8: (*промывка чистой водой после дезинфекции, ожидание протока на возврате*)
  PastPrev:=Step;
  q_SP_P1:=i_PumpCapacity;
  StepBackPump:=1; (*включен возврат и контроль возврата*)

  Start_Control_Q4 := TRUE; (*контроль потока в танк возвратной воды Q4 *)
  ModeControl_Q5 := 2; (*поддержание уровня в цирк баке при промывке и вытесн через цирк бак, контроль насоса Р1*)

  IF Return_OK THEN (*возврта в норме*)
      T_Process.PT:=DINT_TO_TIME(i_TimeSwill*60000);
     Step:=9;
  END_IF;

  q_VisuMode:=19;

9: (*промывка чистой водой после дезинфекции - отсчет времени*)
  PastPrev:=Step;
  q_SP_P1:=i_PumpCapacity;
  StepBackPump:=1; (*включен возврат и контроль возврата*)

  Start_Control_Q4 := TRUE; (*контроль потока в танк возвратной воды Q4 *)
  ModeControl_Q5 := 2; (*поддержание уровня в цирк баке при промывке и вытесн через цирк бак, контроль насоса Р1*)


     (*расчет времени для визуализ*)
    q_Vis_tim_Process := TRUE; (*визуализация полей времени*)
    Last_Time_min := (TIME_TO_DINT(T_Process.PT-T_Process.ET))/60000 ;
    Last_Time_sec := (TIME_TO_DINT(T_Process.PT-T_Process.ET)/1000) - Last_Time_min * 60 ;

   T_Process.in:=TRUE;
   IF T_Process.Q THEN
      T_Process.in:=FALSE;
      Step:=10;
   END_IF;

  q_VisuMode:=19;

10: (*опустошение цирк бака*)
  PastPrev:=Step;
  q_VA51:=TRUE;
  q_P1:=TRUE;
  q_SP_P1:=i_PumpCapacity;
  StepBackPump:=1; (*включен возврат и контроль возврата*)

  Start_Control_Q4 := TRUE; (*контроль потока в танк возвратной воды Q4 *)


    IF (T_LSL_off.Q AND NOT i_LSM) THEN  (*циркуляционный бак пустой*)
      StepBackPump:=3;
      T_Delay.IN:= FALSE;
      Step:=11 ;
    END_IF;

  q_VisuMode:=4;

11: (*откачка из маршрута*)
  PastPrev:=Step;
  StepBackPump:=3; (*откачка из маршрута*)

  T_Delay.PT:=DINT_TO_TIME(i_TimeDelay*1000); (*задержка закрытия клапана*)
  T_Delay.IN:=TRUE;
  q_VA51:=NOT T_Delay.Q ;

  Start_Control_Q4 := TRUE; (*контроль потока в танк возвратной воды Q4 *)


      IF EndReturn  THEN (*докачали из маршрута*)
          T_Delay.IN:= FALSE;
         StepBackPump:=0; (*выключить возврат и контроль возврата*)
         Step:=12;
      END_IF;

  q_VisuMode:=4;

12: (*выполнено*)
  q_VisuMode:=1;
  StepBackPump := 0; (*выключить вовзрат и контроль возврата*)




(*-----------------авария----------------*)
30: (*авария*)
       q_VisuMode:=11;
       q_Red:=TRUE;
       q_Sirena :=TRUE;
       T_Process.IN := FALSE; (*остановка таймера процесса*)
       IF AlarmReset AND (PastPrev=4 OR PastPrev=9)  THEN
          T_Process.PT := DINT_TO_TIME(Last_Time_min*60000 + Last_Time_sec*1000);  (*уставка для таймера  в случае выхода в аварию*)
          Step := PastPrev;
       ELSIF AlarmReset AND PastPrev<>4 AND PastPrev<>9 THEN
          Step := PastPrev;
       END_IF;

(*-----------------пауза----------------*)
35: (*пауза*)
       q_VisuMode:=12;
       q_Yellow:=TRUE;
       T_Process.IN := FALSE; (*остановка таймера процесса*)
       IF NOT i_Pause AND (PastPrev=4 OR PastPrev=9)  THEN
          T_Process.PT := DINT_TO_TIME(Last_Time_min*60000 + Last_Time_sec*1000);  (*уставка для таймера  в случае выхода в аварию*)
          Step := PastPrev;
       ELSIF NOT i_Pause AND PastPrev<>4 AND PastPrev<>9 THEN
          Step := PastPrev;
       END_IF;

(*-----------------пауза - не готов маршрут----------------*)
36: (*пауза*)
       q_VisuMode:=18;
       q_Yellow:=TRUE;
       T_Process.IN := FALSE; (*остановка таймера процесса*)
       IF i_Ready_Route AND (PastPrev=4 OR PastPrev=9)  THEN
          T_Process.PT := DINT_TO_TIME(Last_Time_min*60000 + Last_Time_sec*1000);  (*уставка для таймера  в случае выхода в аварию*)
          Step := PastPrev;
       ELSIF i_Ready_Route AND PastPrev<>4 AND PastPrev<>9 THEN
          Step := PastPrev;
       END_IF;


 END_CASE;

(*блок поддержания уровня в циркуляционном баке во время мойки и при откачке*)
Control_Q5(
	i_P1:= q_P1,
	i_VA551:= q_VA551 ,
	i_VA11:= q_VA11 ,
	i_VA51:= q_VA51 ,
	i_LSL:= i_LSL ,
	i_LSM:= i_LSM ,
	i_LSH:= i_LSH ,
	i_RouteType:= i_RouteType,
	i_Time_LSH_on:= i_Time_LSH_on ,
	i_Time_LSM_on:= i_Time_LSM_on ,
	i_Time_LSM_off:= i_Time_LSM_off ,
	i_Time_LSL_off:= i_Time_LSL_off ,
	i_TimeDelay:= i_TimeDelay ,
	i_ModeControl_Q5:= ModeControl_Q5 ,
	i_StepBackPump:= StepBackPump ,
	q_P1=> q_P1 ,
	q_VA551=> q_VA551 ,
	q_VA11=> q_VA11 ,
	q_VA51=> q_VA51 ,
	q_Alarm_Empty_Q5=> q_Alarm_Empty_Q5 ,
	q_StepBackPump=> StepBackPump);

(*блок контроля и управления возвратом моющих средств*)
Return_Flow(
	i_AlarmPause:= (Step>=30),  (*в аварии или в паузе мойки или неготовности маршрута*)
	i_FS:= i_FS ,
	i_StepBackPump:= StepBackPump ,
	i_RouteType:= i_RouteType ,
	i_Current_VolumeFC11:= i_Current_VolumeFC11 ,
	i_TimeDelayRetPump:= i_TimeDelayRetPump ,
	i_TimeDelayRetFlow:= i_TimeDelayRetFlow ,
	i_TimeAlarmBackFlow:= i_TimeAlarmBackFlow ,
	q_BackPump=> q_BackPump ,
	q_AlarmBackFlow=> q_AlarmBackFlow ,
	q_EndReturn=>EndReturn  ,
      q_Return_OK=>Return_OK ,
	q_ZeroCount_FC11=> q_ZeroCount_FC11 ,
	q_FC11_start=> q_FC11_start );

(*блок контроля потока в танк возвратной воды Q4*)
Control_Q4(
	i_Start:= Start_Control_Q4 ,
	i_Block_Q4_in:= i_Block_Q4_in ,
	i_VA401:= q_VA401 ,
	i_VA541:= q_VA541 ,
	i_TimeDelay:= i_TimeDelay ,
	q_VA401=> q_VA401 ,
	q_VA541=> q_VA541);


T_Process();
T_Delay();
T_LSH_on (IN:=i_LSH,     PT:=DINT_TO_TIME(i_Time_LSH_on*1000));
T_LSM_on (IN:=i_LSM,     PT:=DINT_TO_TIME(i_Time_LSM_on*1000));
T_LSM_off(IN:=NOT i_LSM, PT:=DINT_TO_TIME(i_Time_LSM_off*1000));
T_LSL_off(IN:=NOT i_LSL, PT:=DINT_TO_TIME(i_Time_LSL_off*1000));
END_FUNCTION_BLOCK

(* POU Inputs, ST *)
PROGRAM Inputs  (*блок масштабирования и обработки аналоговых величин*)
VAR
(*-----общие----*)
	fb_TE2  :AnScaling;
	fb_TE3  :AnScaling;
	fb_LE1  :AnScaling;
	fb_LE2  :AnScaling;
	fb_LE3  :AnScaling;
	fb_LE4  :AnScaling;
	fb_TE4  :AnScaling;

(*---контур 1---*)
	fb_TE11:AnScaling;
	fb_PE1  :AnScaling;
	fb_FE1  :AnScaling;
	fb_QE1  :AnScaling;
	fb_TE21 :AnScaling;

(*---контур 2---*)
	fb_TE12 :AnScaling;
	fb_PE2  :AnScaling;
	fb_FE2  :AnScaling;
	fb_QE2  :AnScaling;
	fb_TE22 :AnScaling;


(*расчет концентрации растворов*)
    Conc_C1 :Concentrat_Mode;
    Conc_C2 :Concentrat_Mode;


END_VAR
(*-----------Общие датчики-------------*)
fb_TE2(
	i_IW_an:=		TE2_i ,
	i_SensorType:=	1 ,
	i_An_Scale:=	An_Scale_TE2 ,
	q_Error=>		Error_TE2 ,
	q_LE=>			i_TE2 );

fb_TE3(
	i_IW_an:=		TE3_i ,
	i_SensorType:=	1 ,
	i_An_Scale:=	An_Scale_TE3 ,
	q_Error=>		Error_TE3 ,
	q_LE=>			i_TE3 );

fb_LE1(
	i_IW_an:=		LE1_i ,
	i_SensorType:=	0 ,
	i_An_Scale:=	An_Scale_LE1 ,
	q_Error=>		Error_LE1 ,
	q_LE=>			i_LE1 );

fb_LE2(
	i_IW_an:=		LE2_i ,
	i_SensorType:=	0 ,
	i_An_Scale:=	An_Scale_LE2 ,
	q_Error=>		Error_LE2 ,
	q_LE=>			i_LE2 );

fb_LE3(
	i_IW_an:=		LE3_i ,
	i_SensorType:=	0 ,
	i_An_Scale:=	An_Scale_LE3 ,
	q_Error=>		Error_LE3 ,
	q_LE=>			i_LE3 );



(*раскомментировать при использовании танка возвратной воды Q4*)
(*
fb_LE4(
	i_IW_an:=		LE4_i ,
	i_SensorType:=	0 ,
	i_An_Scale:=	An_Scale_LE4 ,
	q_Error=>		Error_LE4 ,
	q_LE=>			i_LE4 );

fb_TE4(
	i_IW_an:=		TE4_i ,
	i_SensorType:=	1 ,
	i_An_Scale:=	An_Scale_TE4 ,
	q_Error=>		Error_TE4 ,
	q_LE=>			i_TE4 );

*)

(*------------------------------Контур 1---------------------------*)

fb_TE11(
	i_IW_an:=		TE11_i ,
	i_SensorType:=	1 ,
	i_An_Scale:=	An_Scale_TE11 ,
	q_Error=>		Error_TE11 ,
	q_LE=>			i_TE11);

fb_PE1(
	i_IW_an:=		PE1_i ,
	i_SensorType:=	1 ,
	i_An_Scale:=	An_Scale_PE1 ,
	q_Error=>		Error_PE1 ,
	q_LE=>			i_PE1 );
IF i_PE1<0 THEN
   i_PE1:=0;
END_IF;

fb_FE1(
	i_IW_an:=		FE1_i ,
	i_SensorType:=	1 ,
	i_An_Scale:=	An_Scale_FE1 ,
	q_Error=>		Error_FE1 ,
	q_LE=>			i_FE1 );


fb_QE1(
	i_IW_an:=		QE1_i ,
	i_SensorType:=	1 ,
	i_An_Scale:=	An_Scale_QE1 ,
	q_Error=>		Error_QE1 ,
	q_LE=>			i_QE1 );


fb_TE21(
	i_IW_an:=		TE21_i ,
	i_SensorType:=	1 ,
	i_An_Scale:=	An_Scale_TE21 ,
	q_Error=>		Error_TE21 ,
	q_LE=>			i_TE21);



(*------------------------------Контур 2---------------------------*)
fb_TE12(
	i_IW_an:=		TE12_i ,
	i_SensorType:=	1 ,
	i_An_Scale:=	An_Scale_TE12 ,
	q_Error=>		Error_TE12 ,
	q_LE=>			i_TE12);


fb_PE2(
	i_IW_an:=		PE2_i ,
	i_SensorType:=	1 ,
	i_An_Scale:=	An_Scale_PE2 ,
	q_Error=>		Error_PE2 ,
	q_LE=>			i_PE2 );
IF i_PE2<0 THEN
   i_PE2:=0;
END_IF;

fb_FE2(
	i_IW_an:=		FE2_i ,
	i_SensorType:=	1 ,
	i_An_Scale:=	An_Scale_FE2 ,
	q_Error=>		Error_FE2 ,
	q_LE=>			i_FE2 );

fb_QE2(
	i_IW_an:=		QE2_i ,
	i_SensorType:=	1 ,
	i_An_Scale:=	An_Scale_QE2 ,
	q_Error=>		Error_QE2 ,
	q_LE=>			i_QE2 );

fb_TE22(
	i_IW_an:=		TE22_i ,
	i_SensorType:=	1 ,
	i_An_Scale:=	An_Scale_TE22 ,
	q_Error=>		Error_TE22 ,
	q_LE=>			i_TE22);


(*--------------Расчет концентрации растворов------------*)
Conc_C1(
	i_QE:=i_QE1 ,
	i_TE:=i_TE21 ,
	i_ModeQE:=ModeQE_C1 ,
	q_QE_priv=>QE1_priv ,
	q_QE=>QE1 );

Conc_C2(
	i_QE:=i_QE2 ,
	i_TE:=i_TE22 ,
	i_ModeQE:=ModeQE_C2 ,
	q_QE_priv=>QE2_priv ,
	q_QE=>QE2 );
END_PROGRAM

(* POU Concentrat_Mode, ST *)
FUNCTION_BLOCK Concentrat_Mode
VAR_INPUT
	i_QE		: REAL;
	i_TE		: REAL;
	i_ModeQE	: INT;
END_VAR
VAR_OUTPUT
	q_QE_priv	: REAL;
	q_QE		: REAL;

END_VAR
VAR
END_VAR
CASE i_ModeQE OF    (*выбор пересчета по контуру*)

0:(*-------------Расчет концентрации щелочи-----------------*)
q_QE_priv:=i_QE/(1+Koef_tempAlk*(i_TE-Temp_etalonAlk));  (*приведение проводимости к эталонной*)
q_QE := 0.5+(q_QE_priv-QE_null_Alk)/Psi_Alk;   (*расчет концентрации %*)

1:(*-------------Расчет концентрации кислоты-----------------*)
q_QE_priv:=i_QE/(1+Koef_tempAcid*(i_TE-Temp_etalonAcid));  (*приведение проводимости к эталонной*)
q_QE := 0.5+(q_QE_priv-QE_null_Acid)/Psi_Acid;   (*расчет концентрации %*)

END_CASE;

IF q_QE_priv<0 THEN
   q_QE_priv:=0;
END_IF;


IF q_QE<0 THEN
   q_QE:=0;
END_IF;
END_FUNCTION_BLOCK

(* POU AlarmReaction, ST *)
PROGRAM AlarmReaction
VAR
	T_PS   :TON;      (*таймер аварии сжатого воздуха*)
	T_FE11 :TON;      (*таймер аварии протока на подаче*)
	T_FE12 :TON;      (*таймер аварии протока на подаче*)

END_VAR
(*авария низкого давления сжатого воздуха с таймером*)
   T_PS.IN := NOT PS1_i;
IF T_PS.Q THEN
  	Alarm_PS := TRUE;
END_IF;
IF PS1_i AND Alarm_PS AND AlarmReset THEN
   Alarm_PS := FALSE;
END_IF;
T_PS(PT:=T#3s);

(*авария макс давления PE1*)
IF i_PE1>MaxPressure_C1 THEN
   Alarm_PE1 := TRUE;
ELSIF i_PE1<(MaxPressure_C1-2.0) AND  Alarm_PE1 AND AlarmReset THEN
   Alarm_PE1 := FALSE;
END_IF;

(*авария макс давления PE2*)
IF i_PE2>MaxPressure_C2 THEN
   Alarm_PE2 := TRUE;
ELSIF i_PE2<(MaxPressure_C2-2.0) AND  Alarm_PE2 AND AlarmReset THEN
   Alarm_PE2 := FALSE;
END_IF;


(*аварийный стоп*)
IF NOT AlarmStop_i THEN
   Alarm_Stop:=TRUE;
ELSIF Alarm_Stop AND AlarmReset THEN
   Alarm_Stop:=FALSE;
END_IF;

(*нет протока на подаче контура 1*)
T_FE11.IN:=w_qDevice_C1.P1 AND SP_P1>1500 AND i_FE1<1500;
IF T_FE11.Q THEN
   Alarm_FE11:=TRUE;
END_IF;
T_FE11(PT:= DINT_TO_TIME(Time_Alarm_FE*1000));

(*нет протока на подаче контура 2*)
T_FE12.IN:=w_qDevice_C2.P1 AND SP_P2>1500 AND i_FE2<1500;
IF T_FE12.Q THEN
   Alarm_FE12:=TRUE;
END_IF;
T_FE12(PT:= DINT_TO_TIME(Time_Alarm_FE*1000));



IF AlarmReset THEN
   Alarm_FE11:=FALSE;
   Alarm_FE12:=FALSE;
   AlarmBackFlow_C1:=FALSE;
   AlarmBackFlow_C2:=FALSE;
   HeatingAlarm_C1:=FALSE;
   HeatingAlarm_C2:=FALSE;
   CondAlarm_C1:=FALSE;
   CondAlarm_C2:=FALSE;
   Alarm_Empty_Q5:=FALSE;
   Alarm_Empty_Q6:=FALSE;
END_IF;


(*аварийный уровень в баке концентрата кислоты*)
IF NOT LS81_i THEN
   Alarm_LS81:= TRUE;
ELSE
   Alarm_LS81:= FALSE;
END_IF;
(*низкий уровень в баке концентрата кислоты*)
IF NOT LS82_i THEN
   Alarm_LS82:= TRUE;
ELSE
   Alarm_LS82:= FALSE;
END_IF;

(*аварийный уровень в баке концентрата щелочи*)
IF NOT LS71_i THEN
   Alarm_LS71:= TRUE;
ELSE
   Alarm_LS71:= FALSE;
END_IF;
(*низкий уровень в баке концентрата щелочи*)
IF NOT LS72_i THEN
   Alarm_LS72:= TRUE;
ELSE
   Alarm_LS72:= FALSE;
END_IF;



(*минимальный уровень в танке чистой воды*)
IF i_LE1<MinAlarmLevel_Q1 THEN
   Alarm_MinLev_Q1:=TRUE;
ELSIF Alarm_MinLev_Q1 AND i_LE1>(MinAlarmLevel_Q1+5.0) AND AlarmReset THEN
   Alarm_MinLev_Q1:=FALSE;
END_IF;

(*минимальный уровень в танке щелочи*)
IF i_LE2<MinAlarmLevel_Q2 THEN
   Alarm_MinLev_Q2:=TRUE;
ELSIF Alarm_MinLev_Q2 AND i_LE2>(MinAlarmLevel_Q2+5.0) AND AlarmReset THEN
   Alarm_MinLev_Q2:=FALSE;
END_IF;

(*минимальный уровень в танке кислоты*)
IF i_LE3<MinAlarmLevel_Q3 THEN
   Alarm_MinLev_Q3:=TRUE;
ELSIF Alarm_MinLev_Q3 AND i_LE3>(MinAlarmLevel_Q3+5.0) AND AlarmReset THEN
   Alarm_MinLev_Q3:=FALSE;
END_IF;
END_PROGRAM

(* POU DeviceControl, ST *)
PROGRAM DeviceControl
VAR
	Step_Q1		: INT;

(*---блоки управления механизмами--*)
	fb_VA1   	:Valve;
(*контур 1*)
	fb_VA541 	:Valve;
	fb_VA401 	:Valve;
	fb_VA201 	:Valve;
	fb_VA301 	:Valve;
	fb_VA41  	:Valve;
	fb_VA11  	:Valve;
	fb_VA21  	:Valve;
	fb_VA31  	:Valve;
	fb_VA5 		:Valve;
	fb_VA501 	:Valve;
	fb_VA51  	:Valve;
	fb_VA511 	:Valve;
	fb_VA521 	:Valve;
	fb_VA531 	:Valve;
	fb_P1    		:Pump;
(*контур 2*)
	fb_VA642 	:Valve;
	fb_VA402 	:Valve;
	fb_VA202 	:Valve;
	fb_VA302 	:Valve;
	fb_VA42  	:Valve;
	fb_VA12  	:Valve;
	fb_VA22  	:Valve;
	fb_VA32  	:Valve;
	fb_VA6 		:Valve;
	fb_VA602 	:Valve;
	fb_VA62  	:Valve;
	fb_VA612 	:Valve;
	fb_VA622 	:Valve;
	fb_VA632 	:Valve;
	fb_P2    		:Pump;

(*-----ПИД-регуляторы-----*)
	PID_VR1  :PID_M;
	PID_VR2  :PID_M;

	PID_P1   :PID_M;
	PID_P2   :PID_M;

END_VAR
(*управление поддержанием уровня чистой воды в Q1*)
CASE Mode_Q1 OF
0:(*автомат*)
 	CASE Step_Q1 OF
  	0:
   		IF i_LE1<=MinLevel_Q1 THEN
      			Step_Q1:=1;
   		END_IF;
  	1:
   		q_VA1:=TRUE;
   		IF i_LE1>=MaxLevel_Q1 THEN
      			Step_Q1:=0;
   		END_IF;
	END_CASE;
  	Man_VA1:=FALSE;
1:(*ручной*)
  	q_VA1:=Man_VA1;
END_CASE;

fb_VA1(
    i_AlarmReset:=AlarmReset ,
	i_VAopen:=NOT VA1_i ,
	i_VAclose:=VA1_i ,
	i_DiagVA:=DiagVA1 ,
	i_SetVA:=q_VA1 ,
	i_TimerPT:=T#8s ,
	q_Alarm=>Alarm_VA1 ,
	q_VA=>VA1_q);
Mode_VA1:=fb_VA1.Mode;


(*----------------------Управление механизмами с контролем состояния-----------------*)

(*---------------------Контур 1------------------------*)
fb_VA541(
    i_AlarmReset:=AlarmReset ,
	i_VAopen:=NOT VA541_i ,
	i_VAclose:=VA541_i ,
	i_DiagVA:=wDiagVA_C1.VA541 ,
	i_SetVA:=w_qDevice_C1.VA541 ,
	i_TimerPT:=T#5s ,
	q_Alarm=>Alarm_VA541 ,
	q_VA=>VA541_q);
Mode_VA541:=fb_VA541.Mode;

(* раскомментировать при использовании танка возвратной воды Q4
fb_VA401(
    i_AlarmReset:=AlarmReset ,
	i_VAopen:=NOT VA401_i ,
	i_VAclose:=VA401_i ,
	i_DiagVA:=wDiagVA_C1.VA401 ,
	i_SetVA:=w_qDevice_C1.VA401 ,
	i_TimerPT:=T#5s ,
	q_Alarm=>Alarm_VA401 ,
	q_VA=>VA401_q);
Mode_VA401:=fb_VA401.Mode;
*)

fb_VA201(
    i_AlarmReset:=AlarmReset ,
	i_VAopen:=NOT VA201_i ,
	i_VAclose:=VA201_i ,
	i_DiagVA:=wDiagVA_C1.VA201 ,
	i_SetVA:=w_qDevice_C1.VA201 ,
	i_TimerPT:=T#5s ,
	q_Alarm=>Alarm_VA201 ,
	q_VA=>VA201_q);
Mode_VA201:=fb_VA201.Mode;

fb_VA301(
    i_AlarmReset:=AlarmReset ,
	i_VAopen:=NOT VA301_i ,
	i_VAclose:=VA301_i ,
	i_DiagVA:=wDiagVA_C1.VA301 ,
	i_SetVA:=w_qDevice_C1.VA301 ,
	i_TimerPT:=T#5s ,
	q_Alarm=>Alarm_VA301 ,
	q_VA=>VA301_q);
Mode_VA301:=fb_VA301.Mode;

(*раскомментировать при использовании танка возвратной воды Q4
fb_VA41(
    i_AlarmReset:=AlarmReset ,
	i_VAopen:=NOT VA41_i ,
	i_VAclose:=VA41_i ,
	i_DiagVA:=wDiagVA_C1.VA41 ,
	i_SetVA:=w_qDevice_C1.VA41 ,
	i_TimerPT:=T#7s ,
	q_Alarm=>Alarm_VA41 ,
	q_VA=>VA41_q);
Mode_VA41:=fb_VA41.Mode;
*)

fb_VA11(
    i_AlarmReset:=AlarmReset ,
	i_VAopen:=NOT VA11_i ,
	i_VAclose:=VA11_i ,
	i_DiagVA:=wDiagVA_C1.VA11 ,
	i_SetVA:=w_qDevice_C1.VA11 ,
	i_TimerPT:=T#7s ,
	q_Alarm=>Alarm_VA11 ,
	q_VA=>VA11_q);
Mode_VA11:=fb_VA11.Mode;

fb_VA21(
    i_AlarmReset:=AlarmReset ,
	i_VAopen:=NOT VA21_i ,
	i_VAclose:=VA21_i ,
	i_DiagVA:=wDiagVA_C1.VA21 ,
	i_SetVA:=w_qDevice_C1.VA21 ,
	i_TimerPT:=T#7s ,
	q_Alarm=>Alarm_VA21 ,
	q_VA=>VA21_q);
Mode_VA21:=fb_VA21.Mode;

fb_VA31(
    i_AlarmReset:=AlarmReset ,
	i_VAopen:=NOT VA31_i ,
	i_VAclose:=VA31_i ,
	i_DiagVA:=wDiagVA_C1.VA31 ,
	i_SetVA:=w_qDevice_C1.VA31 ,
	i_TimerPT:=T#7s ,
	q_Alarm=>Alarm_VA31 ,
	q_VA=>VA31_q);
Mode_VA31:=fb_VA31.Mode;


fb_VA5(
    i_AlarmReset:=AlarmReset ,
	i_VAopen:=NOT VA5_i ,
	i_VAclose:=VA5_i ,
	i_DiagVA:=wDiagVA_C1.VA5 ,
	i_SetVA:=w_qDevice_C1.VA5 ,
	i_TimerPT:=T#8s ,
	q_Alarm=>Alarm_VA5 ,
	q_VA=>VA5_q);
Mode_VA5:=fb_VA5.Mode;

fb_VA501(
    i_AlarmReset:=AlarmReset ,
	i_VAopen:=NOT VA501_i ,
	i_VAclose:=VA501_i ,
	i_DiagVA:=wDiagVA_C1.VA501 ,
	i_SetVA:=w_qDevice_C1.VA501 ,
	i_TimerPT:=T#5s ,
	q_Alarm=>Alarm_VA501 ,
	q_VA=>VA501_q);
Mode_VA501:=fb_VA501.Mode;

fb_VA51(
    i_AlarmReset:=AlarmReset ,
	i_VAopen:=NOT VA51_i ,
	i_VAclose:=VA51_i ,
	i_DiagVA:=wDiagVA_C1.VA51 ,
	i_SetVA:=w_qDevice_C1.VA51 ,
	i_TimerPT:=T#5s ,
	q_Alarm=>Alarm_VA51 ,
	q_VA=>VA51_q);
Mode_VA51:=fb_VA51.Mode;

fb_VA511(
    i_AlarmReset:=AlarmReset ,
	i_VAopen:=NOT VA511_i ,
	i_VAclose:=VA511_i ,
	i_DiagVA:=wDiagVA_C1.VA511 ,
	i_SetVA:=w_qDevice_C1.VA511 ,
	i_TimerPT:=T#5s ,
	q_Alarm=>Alarm_VA511 ,
	q_VA=>VA511_q);
Mode_VA511:=fb_VA511.Mode;

fb_VA521(
    i_AlarmReset:=AlarmReset ,
	i_VAopen:=NOT VA521_i ,
	i_VAclose:=VA521_i ,
	i_DiagVA:=wDiagVA_C1.VA521 ,
	i_SetVA:=w_qDevice_C1.VA521 ,
	i_TimerPT:=T#5s ,
	q_Alarm=>Alarm_VA521 ,
	q_VA=>VA521_q);
Mode_VA521:=fb_VA521.Mode;

fb_VA531(
    i_AlarmReset:=AlarmReset ,
	i_VAopen:=NOT VA531_i ,
	i_VAclose:=VA531_i ,
	i_DiagVA:=wDiagVA_C1.VA531 ,
	i_SetVA:=w_qDevice_C1.VA531 ,
	i_TimerPT:=T#5s ,
	q_Alarm=>Alarm_VA531 ,
	q_VA=>VA531_q);
Mode_VA531:=fb_VA531.Mode;

(*насос подачи *)
fb_P1(
	i_AlarmReset:= AlarmReset ,
	IsV_P:=w_qDevice_C1.P1 ,
	Protect:= NOT ProtectP1_i ,
	SetV_P:=w_qDevice_C1.P1 ,
	Timer_PT:=t#3s ,
	Alarm=>Alarm_P1 ,
	q_P=> P1_q );
Mode_P1:=fb_P1.Mode;


(*---------------------Контур 2------------------------*)

fb_VA642(
    i_AlarmReset:=AlarmReset ,
	i_VAopen:=NOT VA642_i ,
	i_VAclose:=VA642_i ,
	i_DiagVA:=wDiagVA_C2.VA541 ,
	i_SetVA:=w_qDevice_C2.VA541 ,
	i_TimerPT:=T#5s ,
	q_Alarm=>Alarm_VA642 ,
	q_VA=>VA642_q);
Mode_VA642:=fb_VA642.Mode;

(*раскомментировать при использовании танка возвратной воды Q4
fb_VA402(
    i_AlarmReset:=AlarmReset ,
	i_VAopen:=NOT VA402_i ,
	i_VAclose:=VA402_i ,
	i_DiagVA:=wDiagVA_C2.VA401 ,
	i_SetVA:=w_qDevice_C2.VA401 ,
	i_TimerPT:=T#5s ,
	q_Alarm=>Alarm_VA402 ,
	q_VA=>VA402_q);
Mode_VA402:=fb_VA402.Mode;
*)

fb_VA202(
    i_AlarmReset:=AlarmReset ,
	i_VAopen:=NOT VA202_i ,
	i_VAclose:=VA202_i ,
	i_DiagVA:=wDiagVA_C2.VA201 ,
	i_SetVA:=w_qDevice_C2.VA201 ,
	i_TimerPT:=T#5s ,
	q_Alarm=>Alarm_VA202 ,
	q_VA=>VA202_q);
Mode_VA202:=fb_VA202.Mode;

fb_VA302(
    i_AlarmReset:=AlarmReset ,
	i_VAopen:=NOT VA302_i ,
	i_VAclose:=VA302_i ,
	i_DiagVA:=wDiagVA_C2.VA301 ,
	i_SetVA:=w_qDevice_C2.VA301 ,
	i_TimerPT:=T#5s ,
	q_Alarm=>Alarm_VA302 ,
	q_VA=>VA302_q);
Mode_VA302:=fb_VA302.Mode;

(*раскомментировать при использовании танка возвратной воды Q4
fb_VA42(
    i_AlarmReset:=AlarmReset ,
	i_VAopen:=NOT VA42_i ,
	i_VAclose:=VA42_i ,
	i_DiagVA:=wDiagVA_C2.VA41 ,
	i_SetVA:=w_qDevice_C2.VA41 ,
	i_TimerPT:=T#5s ,
	q_Alarm=>Alarm_VA42 ,
	q_VA=>VA42_q);
Mode_VA42:=fb_VA42.Mode;
*)

fb_VA12(
    i_AlarmReset:=AlarmReset ,
	i_VAopen:=NOT VA12_i ,
	i_VAclose:=VA12_i ,
	i_DiagVA:=wDiagVA_C2.VA11 ,
	i_SetVA:=w_qDevice_C2.VA11 ,
	i_TimerPT:=T#5s ,
	q_Alarm=>Alarm_VA12 ,
	q_VA=>VA12_q);
Mode_VA12:=fb_VA12.Mode;

fb_VA22(
    i_AlarmReset:=AlarmReset ,
	i_VAopen:= NOT VA22_i ,
	i_VAclose:= VA22_i ,
	i_DiagVA:=wDiagVA_C2.VA21 ,
	i_SetVA:=w_qDevice_C2.VA21 ,
	i_TimerPT:=T#7s ,
	q_Alarm=>Alarm_VA22 ,
	q_VA=>VA22_q);
Mode_VA22:=fb_VA22.Mode;

fb_VA32(
    i_AlarmReset:=AlarmReset ,
	i_VAopen:=NOT VA32_i ,
	i_VAclose:=VA32_i ,
	i_DiagVA:=wDiagVA_C2.VA31 ,
	i_SetVA:=w_qDevice_C2.VA31 ,
	i_TimerPT:=T#7s ,
	q_Alarm=>Alarm_VA32 ,
	q_VA=>VA32_q);
Mode_VA32:=fb_VA32.Mode;

fb_VA6(
    i_AlarmReset:=AlarmReset ,
	i_VAopen:=NOT VA6_i ,
	i_VAclose:=VA6_i ,
	i_DiagVA:=wDiagVA_C2.VA5 ,
	i_SetVA:=w_qDevice_C2.VA5 ,
	i_TimerPT:=T#8s ,
	q_Alarm=>Alarm_VA6 ,
	q_VA=>VA6_q);
Mode_VA6:=fb_VA6.Mode;

fb_VA602(
    i_AlarmReset:=AlarmReset ,
	i_VAopen:=NOT VA602_i ,
	i_VAclose:=VA602_i ,
	i_DiagVA:=wDiagVA_C2.VA501 ,
	i_SetVA:=w_qDevice_C2.VA501 ,
	i_TimerPT:=T#5s ,
	q_Alarm=>Alarm_VA602 ,
	q_VA=>VA602_q);
Mode_VA602:=fb_VA602.Mode;

fb_VA62(
    i_AlarmReset:=AlarmReset ,
	i_VAopen:=NOT VA62_i ,
	i_VAclose:=VA62_i ,
	i_DiagVA:=wDiagVA_C2.VA51 ,
	i_SetVA:=w_qDevice_C2.VA51 ,
	i_TimerPT:=T#5s ,
	q_Alarm=>Alarm_VA62 ,
	q_VA=>VA62_q);
Mode_VA62:=fb_VA62.Mode;

fb_VA612(
    i_AlarmReset:=AlarmReset ,
	i_VAopen:=NOT VA612_i ,
	i_VAclose:=VA612_i ,
	i_DiagVA:=wDiagVA_C2.VA511 ,
	i_SetVA:=w_qDevice_C2.VA511 ,
	i_TimerPT:=T#5s ,
	q_Alarm=>Alarm_VA612 ,
	q_VA=>VA612_q);
Mode_VA612:=fb_VA612.Mode;

fb_VA622(
    i_AlarmReset:=AlarmReset ,
	i_VAopen:=NOT VA622_i ,
	i_VAclose:=VA622_i ,
	i_DiagVA:=wDiagVA_C2.VA521 ,
	i_SetVA:=w_qDevice_C2.VA521 ,
	i_TimerPT:=T#5s ,
	q_Alarm=>Alarm_VA622 ,
	q_VA=>VA622_q);
Mode_VA622:=fb_VA622.Mode;

fb_VA632(
    i_AlarmReset:=AlarmReset ,
	i_VAopen:=NOT VA632_i ,
	i_VAclose:=VA632_i ,
	i_DiagVA:=wDiagVA_C2.VA531 ,
	i_SetVA:=w_qDevice_C2.VA531 ,
	i_TimerPT:=T#5s ,
	q_Alarm=>Alarm_VA632 ,
	q_VA=>VA632_q);
Mode_VA632:=fb_VA632.Mode;

(* насос подачи *)
fb_P2(
	i_AlarmReset:= AlarmReset ,
	IsV_P:=w_qDevice_C2.P1 ,
	Protect:= NOT  ProtectP2_i ,
	SetV_P:=w_qDevice_C2.P1 ,
	Timer_PT:=t#3s ,
	Alarm=>Alarm_P2 ,
	q_P=> P2_q );
Mode_P2:=fb_P2.Mode;

(*------------------------------------------------------------*)

(*------Управление механизмами без диагностики*)
VE7_q:=q_VE7;
P8_q:=q_P8;
P9_q:=q_P9;




(*======================Управление аналоговыми выходами======================*)

(*===============Клапана пара===============*)
(*защита от перегрева*)
IF (i_TE11>(SP_VR1+20) OR i_TE11>95)  AND w_qDevice_C1.Heating_VR1 THEN (*перегрев*)
   Alarm_TE11:=TRUE;
ELSIF (Alarm_TE11 AND i_TE11<(SP_VR1+3)) OR NOT w_qDevice_C1.Heating_VR1  THEN
   Alarm_TE11:=FALSE;
END_IF;
w_qDevice_C1.VA14:=w_qDevice_C1.Heating_VR1 AND NOT Alarm_TE11 AND w_qDevice_C1.P1 AND i_FE1>(SP_P1*0.5) ;
VA14_q:=w_qDevice_C1.VA14; (*привязка к физ выходу*)

PID_VR1(
	i_Sp:=SP_VR1 ,
	i_PVin:=i_TE11 ,
	i_Gain:=SP_PID_P_VR1 ,
	i_Ti:=SP_PID_I_VR1 ,
       i_Max_Ipart:=100.0 ,
	i_Reset:= NOT w_qDevice_C1.Heating_VR1 OR NOT w_qDevice_C1.P1 OR i_FE1<(SP_P1*0.3) ,
    i_scan_time:=scan_time ,
	q_PV=>q_VR1an );
VR1an_q :=REAL_TO_WORD(q_VR1an*327.67); (*на физический выход*)

(*-----------------------*)
(*защита от перегрева*)
IF (i_TE12>(SP_VR2+20) OR i_TE12>95)  AND w_qDevice_C2.Heating_VR1 THEN (*перегрев*)
   Alarm_TE12:=TRUE;
ELSIF (Alarm_TE12 AND i_TE12<(SP_VR2+3)) OR NOT w_qDevice_C2.Heating_VR1 THEN
   Alarm_TE12:=FALSE;
END_IF;
w_qDevice_C2.VA14:=w_qDevice_C2.Heating_VR1 AND NOT Alarm_TE12 AND w_qDevice_C2.P1 AND i_FE2>(SP_P2*0.5) ;
VA24_q:=w_qDevice_C2.VA14; (*привязка к физ выходу*)

PID_VR2(
	i_Sp:=SP_VR2 ,
	i_PVin:=i_TE12 ,
	i_Gain:=SP_PID_P_VR2 ,
	i_Ti:=SP_PID_I_VR2 ,
       i_Max_Ipart:=100.0 ,
	i_Reset:= NOT w_qDevice_C2.Heating_VR1 OR NOT w_qDevice_C2.P1 OR i_FE2<(SP_P2*0.3) ,
    i_scan_time:=scan_time ,
	q_PV=>q_VR2an );
VR2an_q :=REAL_TO_WORD(q_VR2an*327.67); (*на физический выход*)

(*-----------------------*)



(*===============Управление производительностью насосов =============*)

PID_P1(
	i_Sp:=SP_P1 / An_Scale_FE1.MaxVal * 100.0 ,
	i_PVin:=i_FE1 / An_Scale_FE1.MaxVal * 100.0 ,
	i_Gain:=SP_PID_P_P1 ,
	i_Ti:=SP_PID_I_P1 ,
       i_Max_Ipart:=100.0 ,
	i_Reset:= NOT w_qDevice_C1.P1 OR Error_FE1 ,
	i_scan_time:=scan_time ,
	q_PV=>q_P1an );
P1an_q :=REAL_TO_WORD(q_P1an*327.67); (*на физический выход*)

PID_P2(
	i_Sp:=SP_P2 / An_Scale_FE2.MaxVal * 100.0 ,
	i_PVin:=i_FE2 /An_Scale_FE2.MaxVal * 100.0 ,
	i_Gain:=SP_PID_P_P2 ,
	i_Ti:=SP_PID_I_P2 ,
       i_Max_Ipart:=100.0 ,
	i_Reset:= NOT w_qDevice_C2.P1 OR Error_FE2 ,
	i_scan_time:=scan_time ,
	q_PV=>q_P2an );
P2an_q :=REAL_TO_WORD(q_P2an*327.67); (*на физический выход*)
END_PROGRAM

(* POU Visualisation, ST *)
PROGRAM Visualisation
VAR
	Vis_Pipe_C1:Vis_Pipe;
	Vis_Pipe_C2:Vis_Pipe;

END_VAR
Vis_Pipe_C1(
	i_FS:= FS21_i ,
	i_LSL:= LSL5_i ,
	i_wDevice:= 	w_qDevice_C1 ,
	q_ReturnPipe=> Vis_Pipe_C1_1.0 ,
	q_521_501=> 	Vis_Pipe_C1_1.1 ,
	q_501_301=>	Vis_Pipe_C1_1.2 ,
	q_301_201=>	Vis_Pipe_C1_1.3 ,
	q_201_401=>	Vis_Pipe_C1_1.4 ,
	q_521=>		Vis_Pipe_C1_1.5 ,
	q_501=>		Vis_Pipe_C1_1.6 ,
	q_301=>		Vis_Pipe_C1_1.7 ,
	q_201=>		Vis_Pipe_C1_1.8 ,
	q_401=>		Vis_Pipe_C1_1.9 ,
	q_541=>		Vis_Pipe_C1_1.10 ,
	q_41=>			Vis_Pipe_C1_1.11 ,
	q_11=>			Vis_Pipe_C1_1.12 ,
	q_21=>			Vis_Pipe_C1_1.13 ,
	q_31=>			Vis_Pipe_C1_1.14 ,
	q_51=>			Vis_Pipe_C1_1.15 ,
	q_511=>		Vis_Pipe_C1_2.0 ,
	q_5=>			Vis_Pipe_C1_2.1 ,
	q_Kanaliz=>	Vis_Pipe_C1_2.2 ,
	q_11_21=>		Vis_Pipe_C1_2.3  ,
	q_21_31=>		Vis_Pipe_C1_2.4 ,
	q_31_51=>		Vis_Pipe_C1_2.5 ,
	q_51_P1=>		Vis_Pipe_C1_2.6 ,
	q_P1=>		Vis_Pipe_C1_2.7 ,
	q_531=>		Vis_Pipe_C1_2.8 );

Vis_Pipe_C2(
	i_FS:= FS22_i ,
	i_LSL:= LSL6_i ,
	i_wDevice:= 	w_qDevice_C2 ,
	q_ReturnPipe=> Vis_Pipe_C2_1.0 ,
	q_521_501=> 	Vis_Pipe_C2_1.1 ,
	q_501_301=>	Vis_Pipe_C2_1.2 ,
	q_301_201=>	Vis_Pipe_C2_1.3 ,
	q_201_401=>	Vis_Pipe_C2_1.4 ,
	q_521=>		Vis_Pipe_C2_1.5 ,
	q_501=>		Vis_Pipe_C2_1.6 ,
	q_301=>		Vis_Pipe_C2_1.7 ,
	q_201=>		Vis_Pipe_C2_1.8 ,
	q_401=>		Vis_Pipe_C2_1.9 ,
	q_541=>		Vis_Pipe_C2_1.10 ,
	q_41=>			Vis_Pipe_C2_1.11 ,
	q_11=>			Vis_Pipe_C2_1.12 ,
	q_21=>			Vis_Pipe_C2_1.13 ,
	q_31=>			Vis_Pipe_C2_1.14 ,
	q_51=>			Vis_Pipe_C2_1.15 ,
	q_511=>		Vis_Pipe_C2_2.0 ,
	q_5=>			Vis_Pipe_C2_2.1 ,
	q_Kanaliz=>	Vis_Pipe_C2_2.2 ,
	q_11_21=>		Vis_Pipe_C2_2.3  ,
	q_21_31=>		Vis_Pipe_C2_2.4 ,
	q_31_51=>		Vis_Pipe_C2_2.5 ,
	q_51_P1=>		Vis_Pipe_C2_2.6 ,
	q_P1=>		Vis_Pipe_C2_2.7 ,
	q_531=>		Vis_Pipe_C2_2.8 );





(*отображение полей текущей выполняемой операции в таблице параметров каждого контура*)

w_Step_C1.0 := (Step_C1=2);    (*полоскание возвратной водой*)
w_Step_C1.1 := (Step_C1=4);    (*полоскание свежей водой*)
w_Step_C1.2 := (Step_C1=6);    (*мойка щелочью*)
w_Step_C1.3 := (Step_C1=8);    (*мойка чистой водой 1 после щелочи*)
w_Step_C1.4 := (Step_C1=10);  (*мойка кислотой*)
w_Step_C1.5 := (Step_C1=12);  (*мойка чистой водой 2 после кислоты*)
w_Step_C1.6 := (Step_C1=14);  (*химическая дезинфекция*)
w_Step_C1.7 := (Step_C1=16);  (*термическая дезинфекция*)

w_Step_C2.0 := (Step_C2=2);    (*полоскание возвратной водой*)
w_Step_C2.1 := (Step_C2=4);    (*полоскание свежей водой*)
w_Step_C2.2 := (Step_C2=6);    (*мойка щелочью*)
w_Step_C2.3 := (Step_C2=8);    (*мойка чистой водой 1 после щелочи*)
w_Step_C2.4 := (Step_C2=10);  (*мойка кислотой*)
w_Step_C2.5 := (Step_C2=12);  (*мойка чистой водой 2 после кислоты*)
w_Step_C2.6 := (Step_C2=14);  (*химическая дезинфекция*)
w_Step_C2.7 := (Step_C2=16);  (*термическая дезинфекция*)

(*отображение диcкретных датчиков*)
Vis_FS_K1    := FS21_i;
Vis_LSL_K1  := LSL5_i;
Vis_LSM_K1 := LSM5_i;
Vis_LSH_K1 := LSH5_i;

Vis_FS_K2    := FS22_i;
Vis_LSL_K2  := LSL6_i;
Vis_LSM_K2 := LSM6_i;
Vis_LSH_K2 := LSH6_i;

Vis_ConcAlk_alarm  	:= LS71_i;
Vis_ConcAlk_min	  	:= LS72_i;
Vis_ConcAcid_alarm	:= LS81_i;
Vis_ConcAcid_min		:= LS82_i;

Vis_PS1 := PS1_i;
END_PROGRAM

(* POU Vis_Pipe, ST *)
FUNCTION_BLOCK Vis_Pipe
VAR_INPUT
	i_FS			: BOOL;		(*датчик протока на возврате*)
	i_LSL			: BOOL;		(*датчик нижнего уровня в цирк баке*)
	i_wDevice		:DWORD;	(*слово состояния клапанов*)


END_VAR
VAR_OUTPUT
	q_ReturnPipe: BOOL;
	q_521_501: BOOL;
	q_501_301: BOOL;
	q_301_201: BOOL;
	q_201_401: BOOL;
	q_521: BOOL;
	q_501: BOOL;
	q_301: BOOL;
	q_201: BOOL;
	q_401: BOOL;
	q_541: BOOL;
	q_41: BOOL;
	q_11: BOOL;
	q_21: BOOL;
	q_31: BOOL;
	q_51: BOOL;
	q_511: BOOL;
	q_5: BOOL;
	q_Kanaliz: BOOL;
	q_11_21: BOOL;
	q_21_31: BOOL;
	q_31_51: BOOL;
	q_51_P1: BOOL;
	q_P1: BOOL;
	q_531: BOOL;

END_VAR
VAR
END_VAR
	q_ReturnPipe := (i_wDevice.BackPump OR (i_wDevice.P1 AND NOT i_wDevice.VA531))  AND  i_FS;
	q_521_501 := (i_wDevice.VA501 OR i_wDevice.VA301 OR i_wDevice.VA201 OR i_wDevice.VA401 OR NOT i_wDevice.VA541) AND i_FS ;
	q_501_301 := (i_wDevice.VA301 OR i_wDevice.VA201 OR i_wDevice.VA401 OR NOT i_wDevice.VA541) AND i_FS ;
	q_301_201 := (i_wDevice.VA201 OR i_wDevice.VA401 OR NOT i_wDevice.VA541) AND i_FS ;
	q_201_401 := (i_wDevice.VA401 OR NOT i_wDevice.VA541) AND i_FS ;
	q_521 := i_wDevice.VA521 AND i_FS;
	q_501 := i_wDevice.VA501 AND i_FS;
	q_301 := i_wDevice.VA301 AND i_FS;
	q_201 := i_wDevice.VA201 AND i_FS;
	q_401 := i_wDevice.VA401 AND i_FS;
	q_541 := NOT i_wDevice.VA541 AND i_FS;
	q_41 := i_wDevice.VA41 AND i_wDevice.P1;
	q_11 := i_wDevice.VA11 AND i_wDevice.P1;
	q_21 := i_wDevice.VA21 AND i_wDevice.P1;
	q_31 := i_wDevice.VA31 AND i_wDevice.P1;
	q_51 := i_wDevice.VA51 AND i_wDevice.P1;
	q_511 := i_wDevice.VA511 AND i_LSL ;
	q_5 := i_wDevice.VA5;
	q_Kanaliz := q_511 OR q_541;
	q_11_21 := (i_wDevice.VA41 OR i_wDevice.VA11) AND i_wDevice.P1;
	q_21_31 := (i_wDevice.VA41 OR i_wDevice.VA11 OR i_wDevice.VA21) AND i_wDevice.P1;
	q_31_51 := (i_wDevice.VA41 OR i_wDevice.VA11 OR i_wDevice.VA21 OR i_wDevice.VA31) AND i_wDevice.P1;
	q_51_P1 := (i_wDevice.VA41 OR i_wDevice.VA11 OR i_wDevice.VA21 OR i_wDevice.VA31 OR i_wDevice.VA51) AND i_wDevice.P1;
	q_P1 := i_wDevice.P1 AND (NOT i_wDevice.VA531 OR (i_FS AND i_wDevice.VA521));
	q_531:=i_wDevice.P1 AND NOT i_wDevice.VA531 ;
END_FUNCTION_BLOCK
